// SIMATIC S7-200 project (STEP 7-Micro/WIN), CPU 226 REL 02.01

ORGANIZATION_BLOCK 主程序:OB1
TITLE=程序注释
VAR
I0.0:?;	//  启动按键
I0.1:?;	//  关闭按钮
Q0.0:?;	//  输出
END_VAR
BEGIN
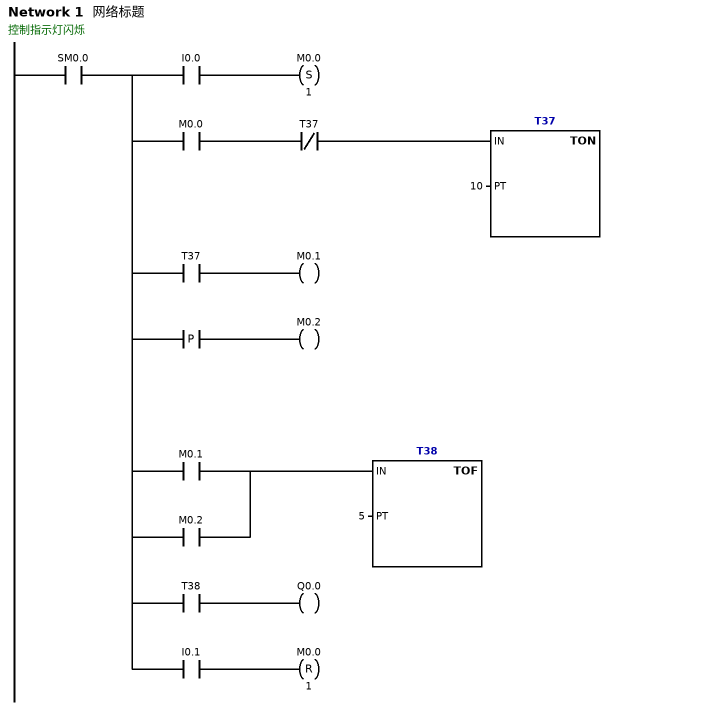
Network 1 // 网络标题
// 控制指示灯闪烁
// (network saved uncompiled; LAD cells follow)
// row 0: c0 -| |- SM0.0 v  c1 -| |- I0.0  c2 -(S) M0.0, 1
// row 1: c0 ^v  c1 -| |- M0.0  c2 -|/|- T37  c3 --  c4 [TON T37 IN:=power@row1, PT:=10]
// row 2: c0 ^v  c4 [box]
// row 3: c0 ^v  c1 -| |- T37  c2 -( ) M0.1
// row 4: c0 ^v  c1 -|P|-  c2 -( ) M0.2
// row 5: c0 ^v
// row 6: c0 ^v  c1 -| |- M0.1 v  c2 --  c3 [TOF T38 IN:=power@row6, PT:=5]
// row 7: c0 ^v  c1 -| |- M0.2 ^  c3 [box]
// row 8: c0 ^v  c1 -| |- T38  c2 -( ) Q0.0
// row 9: c0 ^  c1 -| |- I0.1  c2 -(R) M0.0, 1
END_ORGANIZATION_BLOCK
